{attribute addProperty BoxType "EK1100-0000-0018"}
{attribute addProperty Id "Beckhoff_AT2xxxEK1122Beckhoff_AT2xxxEK1122_A4B15922464805810A_0059_AT2000_5250_0018AT2000_3DCFC8D064080"}
{attribute addProperty CRC "1934353438"}
{attribute addProperty SizeInBites "47120"}
{attribute addProperty SizeInBytes "5890"}
TYPE Beckhoff_AT1xxx_734BE41E EXTENDS EK1100_179A0949 :
STRUCT
	{attribute addProperty Name "Beckhoff_AT2xxxEK1122"}
	Beckhoff_AT2xxxEK1122 : Beckhoff_AT2xxxEK1122_A4B15922;
	{attribute addProperty Name "A_0059_AT2000_5250_0018"}
	A_0059_AT2000_5250_0018 : AT2000_3DCFC8D0;
END_STRUCT
END_TYPE

(* stored: Version 1.2.0.0, ProductVersion 3.1.4024.9
   DUT Beckhoff_AT1xxx_734BE41E: Id {e3eb5ece-0d09-4e1a-9e53-c1b09978a92b} *)
